TYPE "PLCtoMES_RealTimeData"
VERSION : 0.1
   STRUCT
      "P-RealTimeData" : Array[1..64] of "PLCtoMES_ProcessData";
      Reserve { S7_SetPoint := 'True'} : Array[1..100] of Byte;
   END_STRUCT;

END_TYPE

